// SIMATIC S7-200 SMART project (STEP 7-Micro/WIN SMART), CPU ST40

SYMBOL_TABLE 用户定义1
传感器1             I0.0
传感器2             I0.1
传感器3             I0.2
传感器4             I0.3
传感器5             I0.4
传感器6             I0.5
传感器7             I0.6
传感器8             I0.7
END_SYMBOL_TABLE

SYMBOL_TABLE 系统符号
Always_On        SM0.0    // 始终接通
First_Scan_On    SM0.1    // 仅在第一个扫描周期时接通
P0_Config        SMB30    // 组态端口 0 通信：奇偶校验、每个字符的数据位数、波特率和协议
END_SYMBOL_TABLE

SYMBOL_TABLE 表格 3
State            VB5000
SendBuffer       VB5100
RecvBuffer       VB5300
RecvLenth        VW5004
SendLenth        VW5006
SendBufferW      VW5100
RecvBufferW      VW5300
StateConnect     1
StateConnectWait 2
StateTransmit    3
StateTransmitWait 4
StateReceive     5
StateRecvCheck   6
StateDisconnect  7
StateDisconnectWait 8
ExitSwitch       10
SendLenthB       VB5008
END_SYMBOL_TABLE

ORGANIZATION_BLOCK 主程序:OB1
TITLE=程序注释
BEGIN
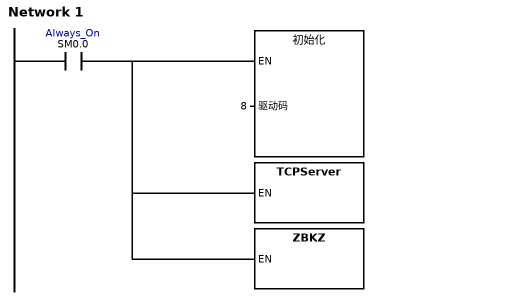
Network 1
LD     Always_On:SM0.0
CALL   初始化:SBR0, 8
CALL   TCPServer:SBR80
CALL   ZBKZ:SBR29
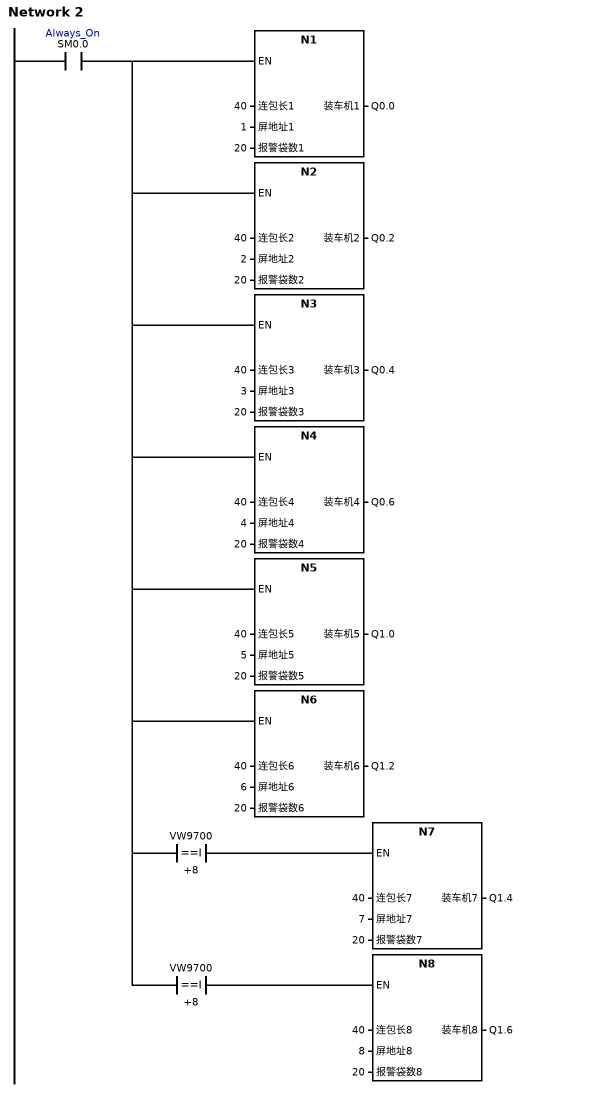
Network 2
LD     Always_On:SM0.0
LPS
CALL   N1:SBR1, 40, 1, 20, Q0.0
CALL   N2:SBR2, 40, 2, 20, Q0.2
CALL   N3:SBR3, 40, 3, 20, Q0.4
CALL   N4:SBR4, 40, 4, 20, Q0.6
CALL   N5:SBR5, 40, 5, 20, Q1.0
CALL   N6:SBR6, 40, 6, 20, Q1.2
AW=    VW9700, +8
CALL   N7:SBR7, 40, 7, 20, Q1.4
LPP
AW=    VW9700, +8
CALL   N8:SBR8, 40, 8, 20, Q1.6
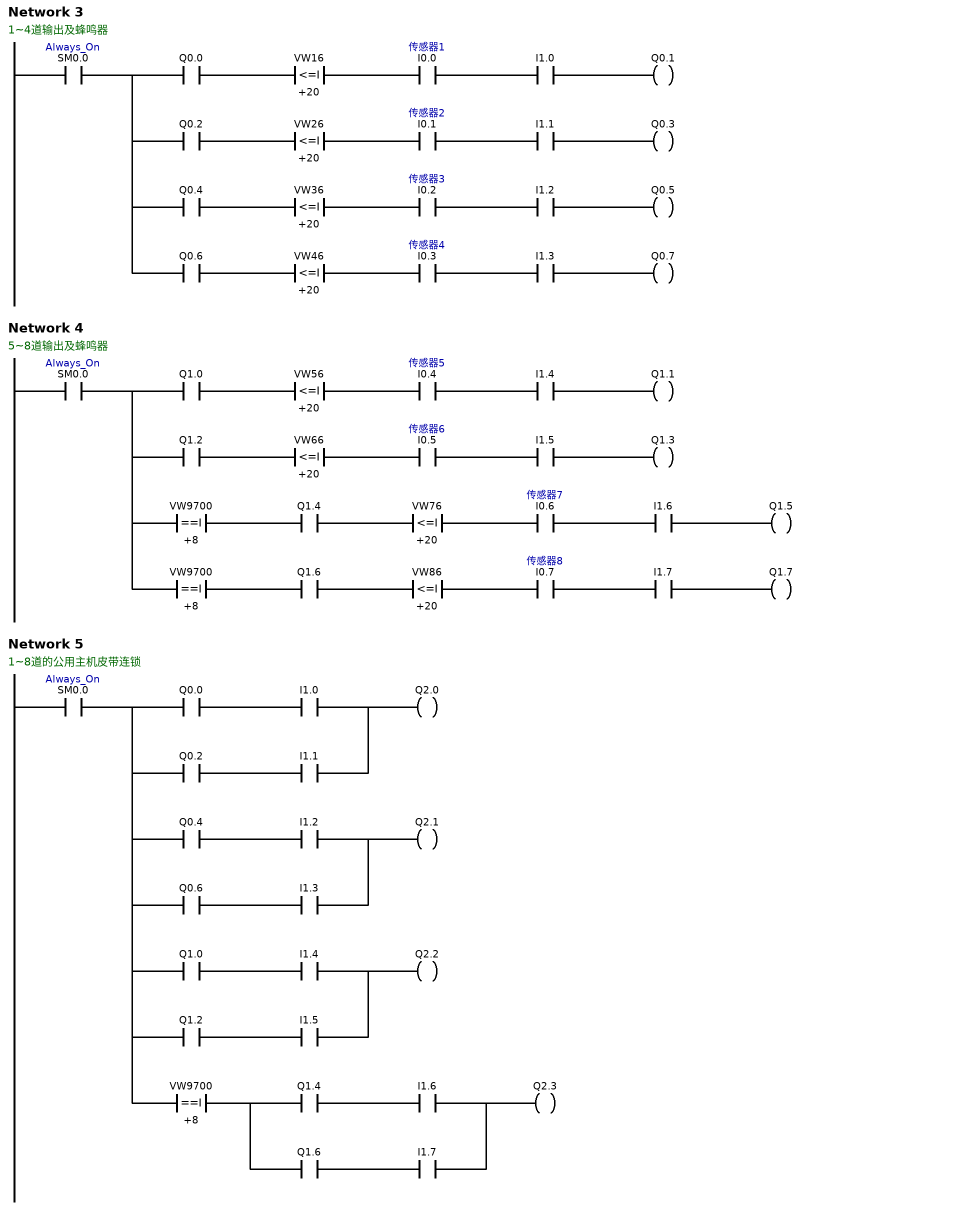
Network 3
// 1~4道输出及蜂鸣器
LD     Always_On:SM0.0
LPS
A      Q0.0
AW<=   VW16, +20
A      传感器1:I0.0
A      I1.0
=      Q0.1
LRD
A      Q0.2
AW<=   VW26, +20
A      传感器2:I0.1
A      I1.1
=      Q0.3
LRD
A      Q0.4
AW<=   VW36, +20
A      传感器3:I0.2
A      I1.2
=      Q0.5
LPP
A      Q0.6
AW<=   VW46, +20
A      传感器4:I0.3
A      I1.3
=      Q0.7
Network 4
// 5~8道输出及蜂鸣器
LD     Always_On:SM0.0
LPS
A      Q1.0
AW<=   VW56, +20
A      传感器5:I0.4
A      I1.4
=      Q1.1
LRD
A      Q1.2
AW<=   VW66, +20
A      传感器6:I0.5
A      I1.5
=      Q1.3
LRD
AW=    VW9700, +8
A      Q1.4
AW<=   VW76, +20
A      传感器7:I0.6
A      I1.6
=      Q1.5
LPP
AW=    VW9700, +8
A      Q1.6
AW<=   VW86, +20
A      传感器8:I0.7
A      I1.7
=      Q1.7
Network 5
// 1~8道的公用主机皮带连锁
LD     Always_On:SM0.0
LPS
LD     Q0.0
A      I1.0
LD     Q0.2
A      I1.1
OLD
ALD
=      Q2.0
LRD
LD     Q0.4
A      I1.2
LD     Q0.6
A      I1.3
OLD
ALD
=      Q2.1
LRD
LD     Q1.0
A      I1.4
LD     Q1.2
A      I1.5
OLD
ALD
=      Q2.2
LPP
AW=    VW9700, +8
LD     Q1.4
A      I1.6
LD     Q1.6
A      I1.7
OLD
ALD
=      Q2.3
END_ORGANIZATION_BLOCK

SUBROUTINE_BLOCK 初始化:SBR0
TITLE=子程序注释
VAR_INPUT
驱动码:WORD;	// LW0 
END_VAR
VAR
temp1:WORD;	// LW2 
temp2:WORD;	// LW4 
END_VAR
BEGIN
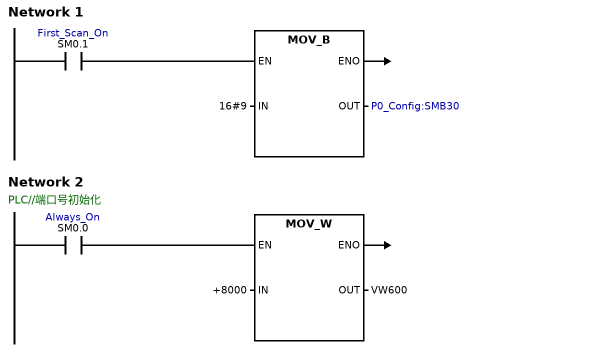
Network 1
// 首次扫描时，
// 初始化自由端口：
// - 选择9600波特
// - 选择8个数据位
// - 选择无校验
// 初始化RCV信息控制字节：
// - RCV被启用
// - 检测到信息字符结束
// - 将空闲行条件检测为
// 信息开始条件。
// 将信息字符结束设为hex OA（换行符）。
// 将空闲行超时设为5毫秒。
// 将最大字符数设为100。
// 为端口0在VB100位置启用带缓冲区的接收方框
LD     First_Scan_On:SM0.1
MOVB   16#9, P0_Config:SMB30
Network 2
// PLC//端口号初始化
LD     Always_On:SM0.0
MOVW   +8000, VW600
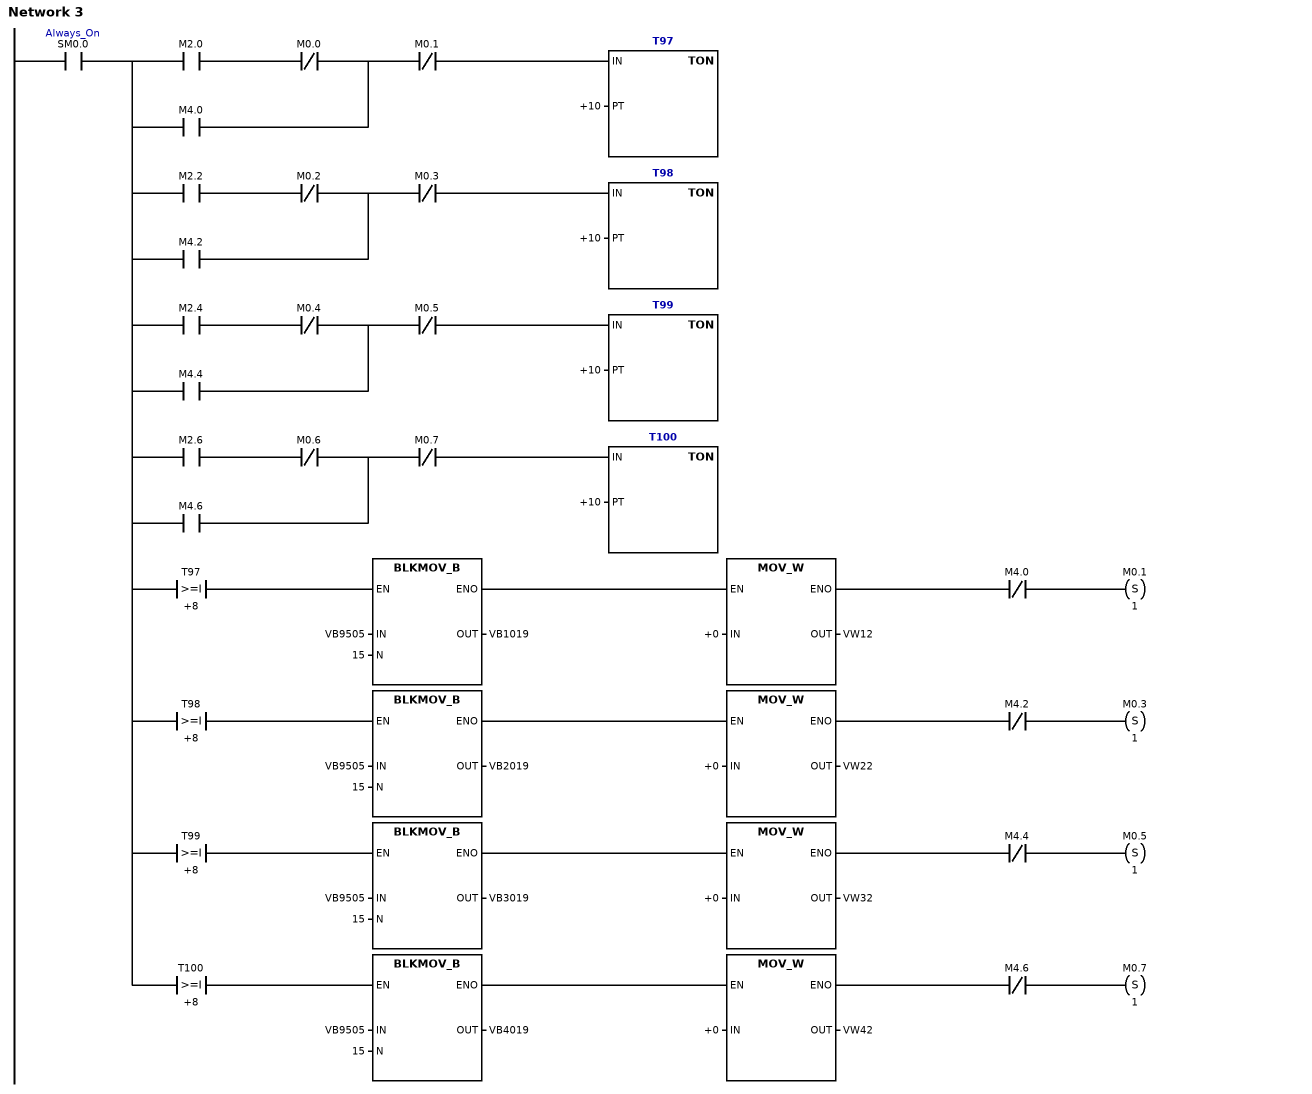
Network 3
LD     Always_On:SM0.0
LPS
LD     M2.0
AN     M0.0
O      M4.0
ALD
AN     M0.1
TON    T97, +10
LRD
LD     M2.2
AN     M0.2
O      M4.2
ALD
AN     M0.3
TON    T98, +10
LRD
LD     M2.4
AN     M0.4
O      M4.4
ALD
AN     M0.5
TON    T99, +10
LRD
LD     M2.6
AN     M0.6
O      M4.6
ALD
AN     M0.7
TON    T100, +10
LPP
LPS
AW>=   T97, +8
BMB    VB9505, VB1019, 15
AENO
MOVW   +0, VW12
AENO
AN     M4.0
S      M0.1, 1
LRD
AW>=   T98, +8
BMB    VB9505, VB2019, 15
AENO
MOVW   +0, VW22
AENO
AN     M4.2
S      M0.3, 1
LRD
AW>=   T99, +8
BMB    VB9505, VB3019, 15
AENO
MOVW   +0, VW32
AENO
AN     M4.4
S      M0.5, 1
LPP
AW>=   T100, +8
BMB    VB9505, VB4019, 15
AENO
MOVW   +0, VW42
AENO
AN     M4.6
S      M0.7, 1
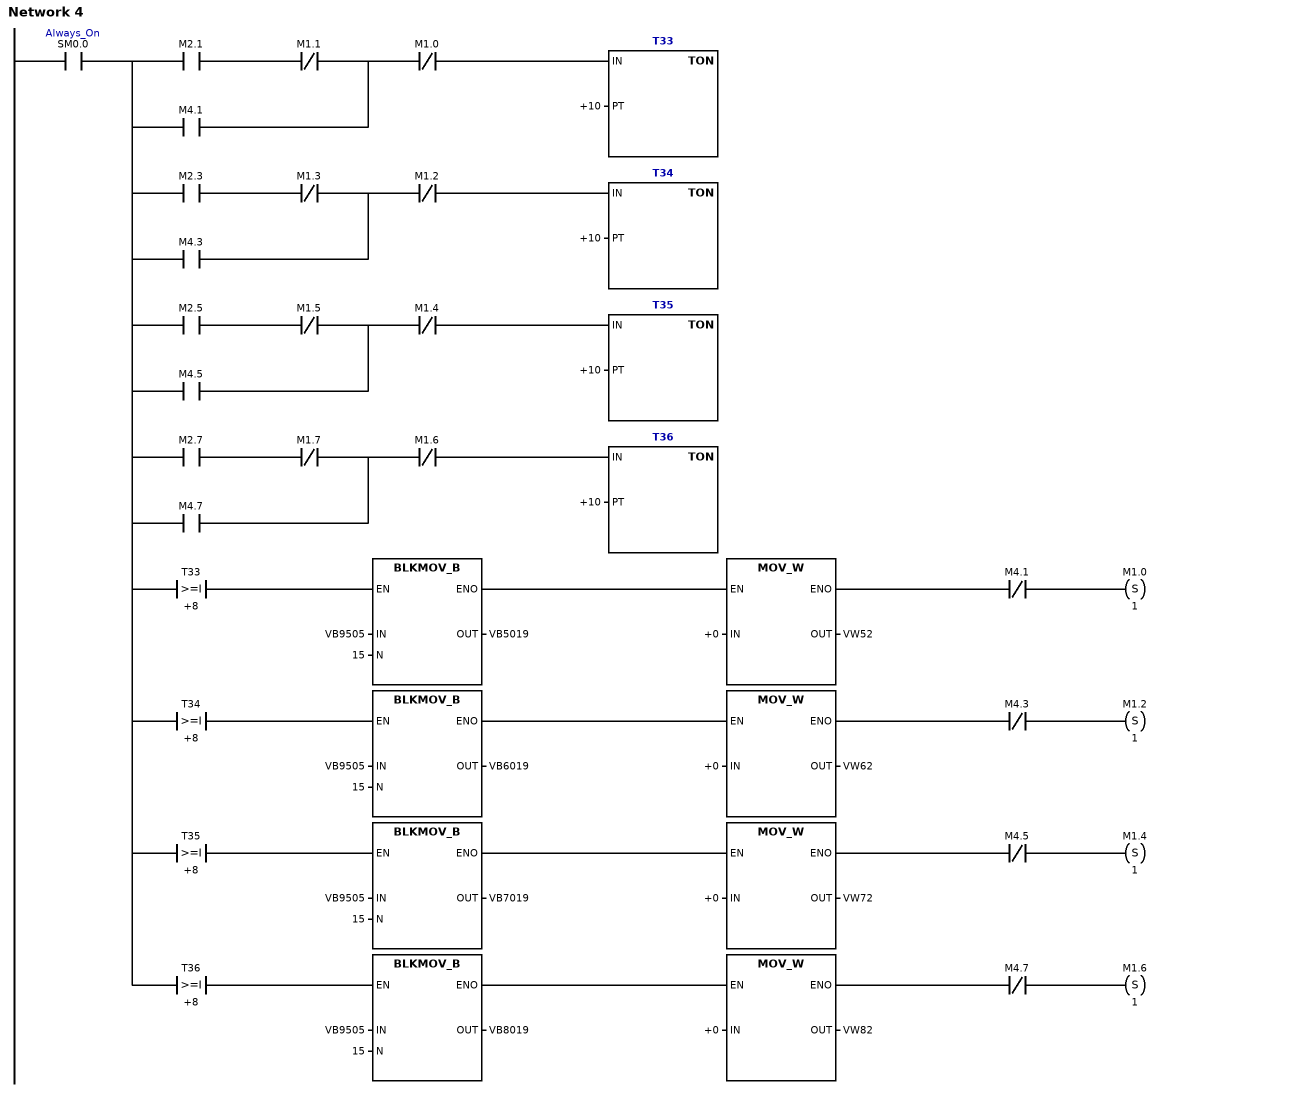
Network 4
LD     Always_On:SM0.0
LPS
LD     M2.1
AN     M1.1
O      M4.1
ALD
AN     M1.0
TON    T33, +10
LRD
LD     M2.3
AN     M1.3
O      M4.3
ALD
AN     M1.2
TON    T34, +10
LRD
LD     M2.5
AN     M1.5
O      M4.5
ALD
AN     M1.4
TON    T35, +10
LRD
LD     M2.7
AN     M1.7
O      M4.7
ALD
AN     M1.6
TON    T36, +10
LPP
LPS
AW>=   T33, +8
BMB    VB9505, VB5019, 15
AENO
MOVW   +0, VW52
AENO
AN     M4.1
S      M1.0, 1
LRD
AW>=   T34, +8
BMB    VB9505, VB6019, 15
AENO
MOVW   +0, VW62
AENO
AN     M4.3
S      M1.2, 1
LRD
AW>=   T35, +8
BMB    VB9505, VB7019, 15
AENO
MOVW   +0, VW72
AENO
AN     M4.5
S      M1.4, 1
LPP
AW>=   T36, +8
BMB    VB9505, VB8019, 15
AENO
MOVW   +0, VW82
AENO
AN     M4.7
S      M1.6, 1
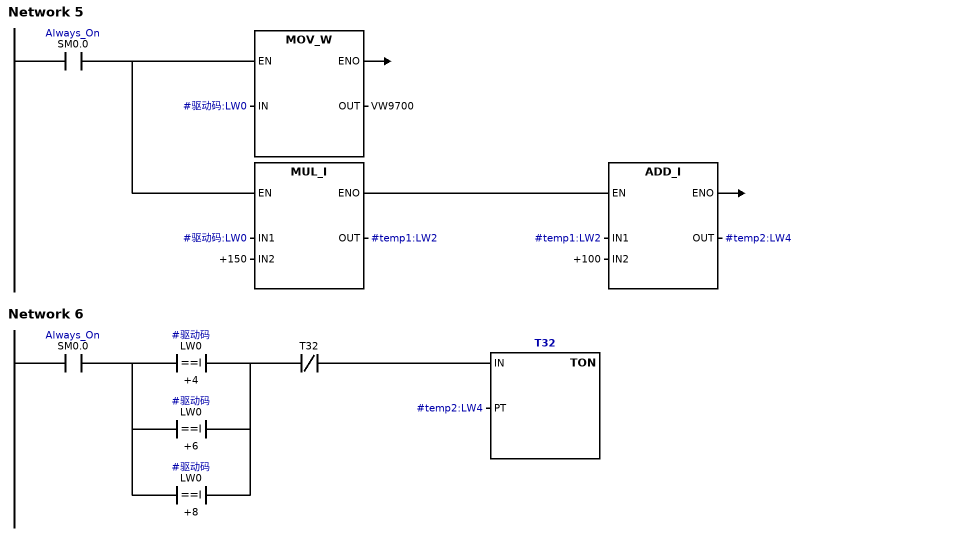
Network 5
LD     Always_On:SM0.0
MOVW   #驱动码:LW0, VW9700
MOVW   #驱动码:LW0, #temp1:LW2
AENO
*I     +150, #temp1:LW2
AENO
MOVW   #temp1:LW2, #temp2:LW4
+I     +100, #temp2:LW4
Network 6
LD     Always_On:SM0.0
LDW=   #驱动码:LW0, +4
OW=    #驱动码:LW0, +6
OW=    #驱动码:LW0, +8
ALD
AN     T32
TON    T32, #temp2:LW4
END_SUBROUTINE_BLOCK

SUBROUTINE_BLOCK N1:SBR1
TITLE=
VAR_INPUT
连包长1:WORD;	// LW0 
屏地址1:BYTE;	// LB2 
报警袋数1:WORD;	// LW3 
END_VAR
VAR_OUTPUT
装车机1:BOOL;	// L5.0 
END_VAR
VAR
总袋数1:WORD;	// LW6 
袋长1:WORD;	// LW8 
已装袋数1:WORD;	// LW10 
剩余袋数1:WORD;	// LW12 
END_VAR
BEGIN
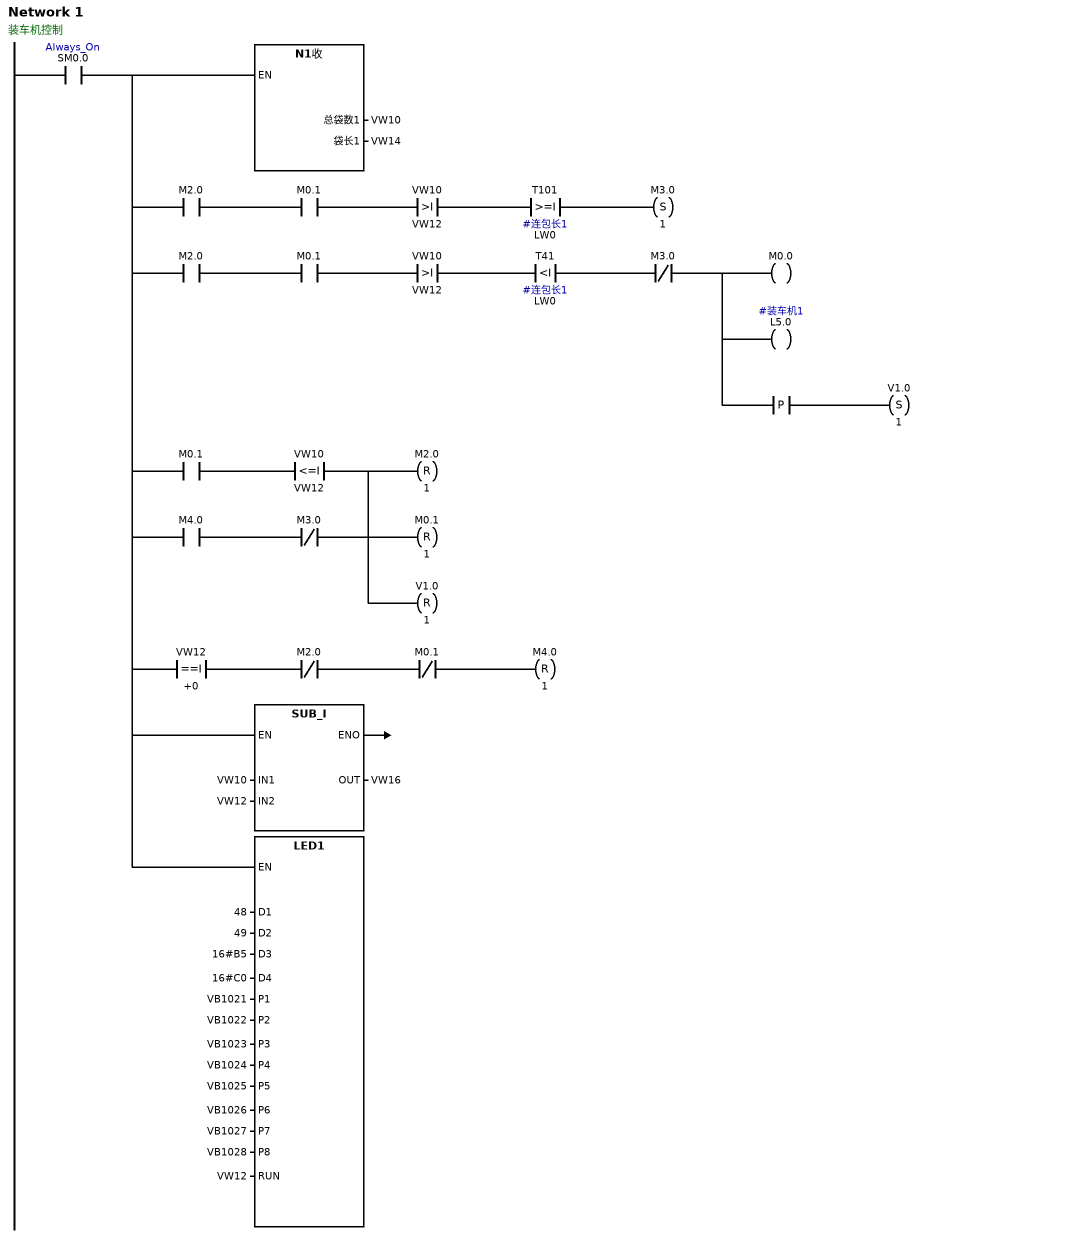
Network 1
// 装车机控制
LD     Always_On:SM0.0
LPS
CALL   N1收:SBR21, VW10, VW14
A      M2.0
A      M0.1
AW>    VW10, VW12
AW>=   T101, #连包长1:LW0
S      M3.0, 1
LRD
A      M2.0
A      M0.1
AW>    VW10, VW12
AW<    T41, #连包长1:LW0
AN     M3.0
=      M0.0
=      #装车机1:L5.0
EU
S      V1.0, 1
LRD
LD     M0.1
AW<=   VW10, VW12
LD     M4.0
AN     M3.0
OLD
ALD
R      M2.0, 1
R      M0.1, 1
R      V1.0, 1
LPP
LPS
AW=    VW12, +0
AN     M2.0
AN     M0.1
R      M4.0, 1
LRD
MOVW   VW10, VW16
-I     VW12, VW16
LPP
CALL   LED1:SBR11, 48, 49, 16#B5, 16#C0, VB1021, VB1022, VB1023, VB1024, VB1025, VB1026, VB1027, VB1028, VW12
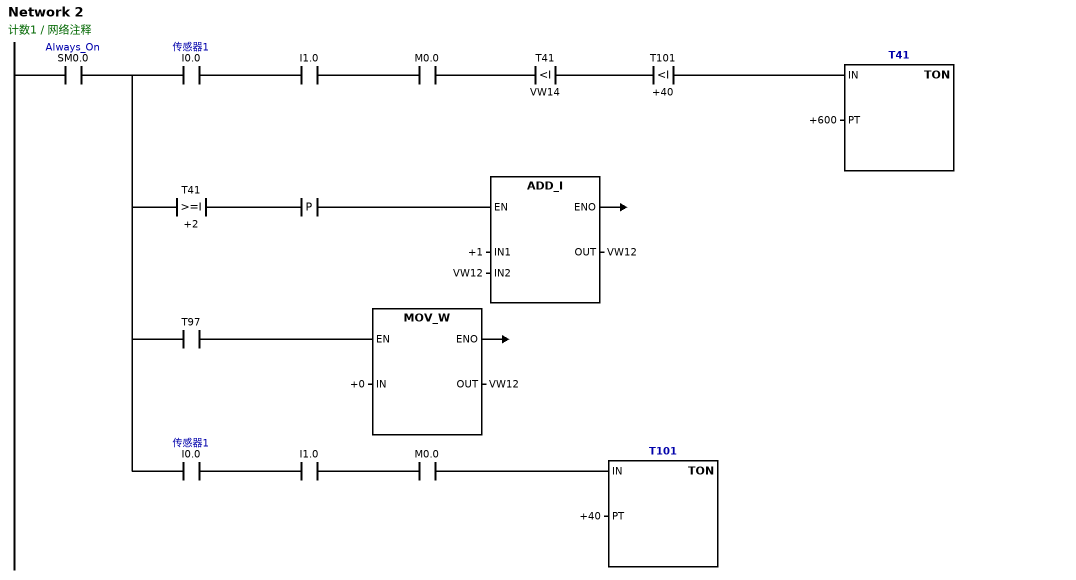
Network 2
// 计数1
// 网络注释
LD     Always_On:SM0.0
LPS
A      传感器1:I0.0
A      I1.0
A      M0.0
AW<    T41, VW14
AW<    T101, +40
TON    T41, +600
LRD
AW>=   T41, +2
EU
+I     +1, VW12
LRD
A      T97
MOVW   +0, VW12
LPP
A      传感器1:I0.0
A      I1.0
A      M0.0
TON    T101, +40
END_SUBROUTINE_BLOCK

SUBROUTINE_BLOCK N2:SBR2
TITLE=
VAR_INPUT
连包长2:WORD;	// LW0 
屏地址2:BYTE;	// LB2 
报警袋数2:WORD;	// LW3 
END_VAR
VAR_OUTPUT
装车机2:BOOL;	// L5.0 
END_VAR
VAR
总袋数2:WORD;	// LW6 
袋长2:WORD;	// LW8 
已装袋数2:WORD;	// LW10 
剩余袋数2:WORD;	// LW12 
END_VAR
BEGIN
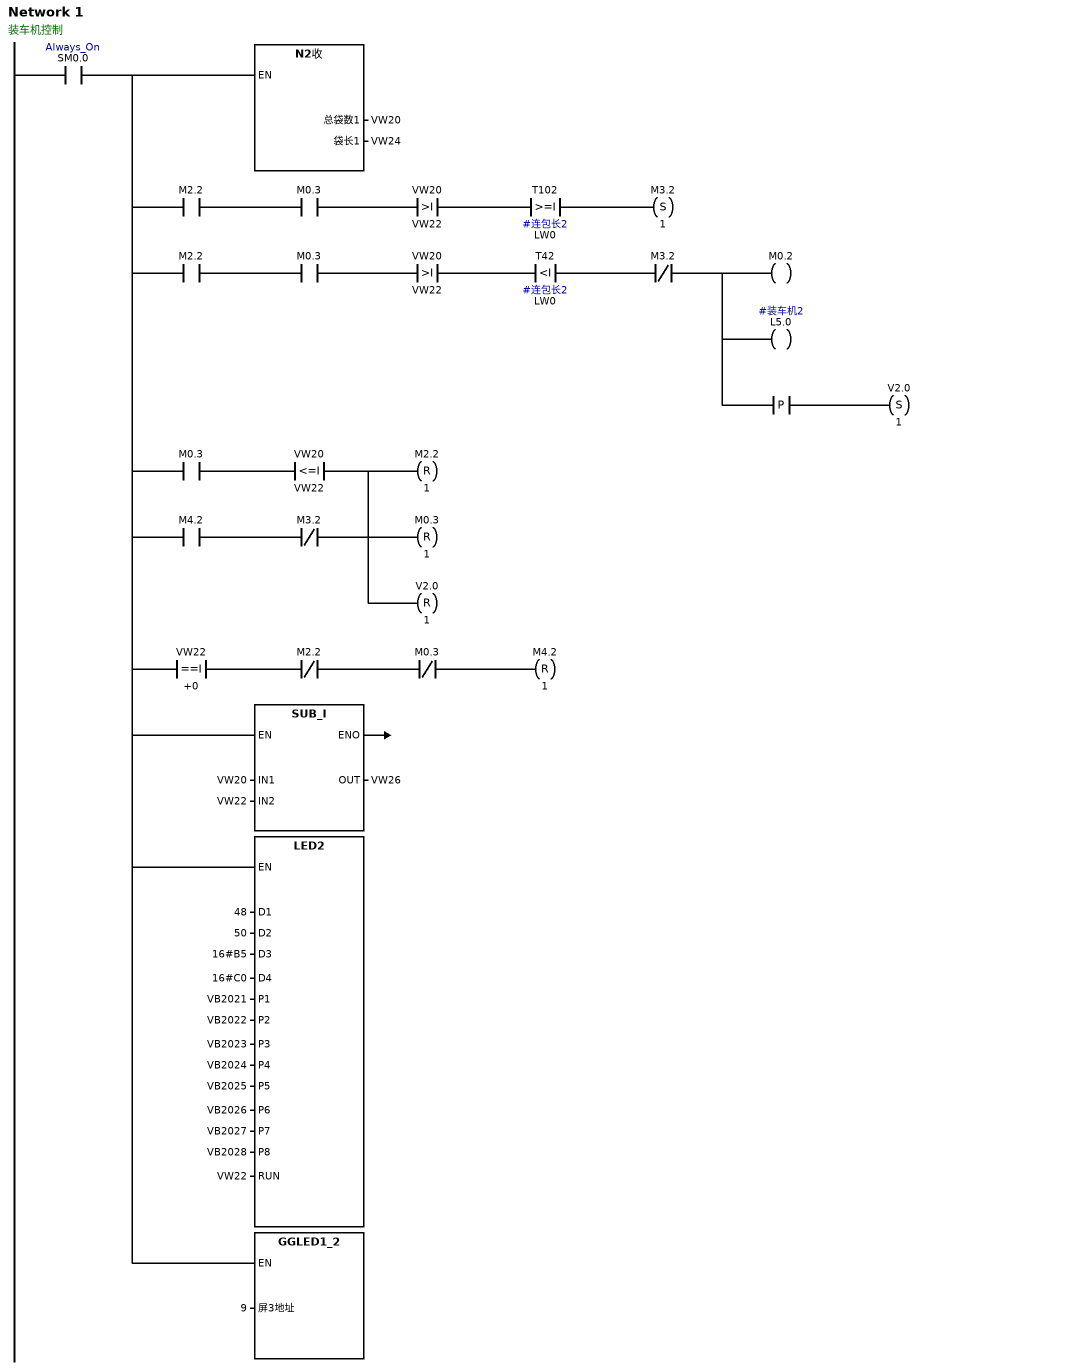
Network 1
// 装车机控制
LD     Always_On:SM0.0
LPS
CALL   N2收:SBR22, VW20, VW24
A      M2.2
A      M0.3
AW>    VW20, VW22
AW>=   T102, #连包长2:LW0
S      M3.2, 1
LRD
A      M2.2
A      M0.3
AW>    VW20, VW22
AW<    T42, #连包长2:LW0
AN     M3.2
=      M0.2
=      #装车机2:L5.0
EU
S      V2.0, 1
LRD
LD     M0.3
AW<=   VW20, VW22
LD     M4.2
AN     M3.2
OLD
ALD
R      M2.2, 1
R      M0.3, 1
R      V2.0, 1
LPP
LPS
AW=    VW22, +0
AN     M2.2
AN     M0.3
R      M4.2, 1
LRD
MOVW   VW20, VW26
-I     VW22, VW26
LRD
CALL   LED2:SBR12, 48, 50, 16#B5, 16#C0, VB2021, VB2022, VB2023, VB2024, VB2025, VB2026, VB2027, VB2028, VW22
LPP
CALL   GGLED1_2:SBR31, 9
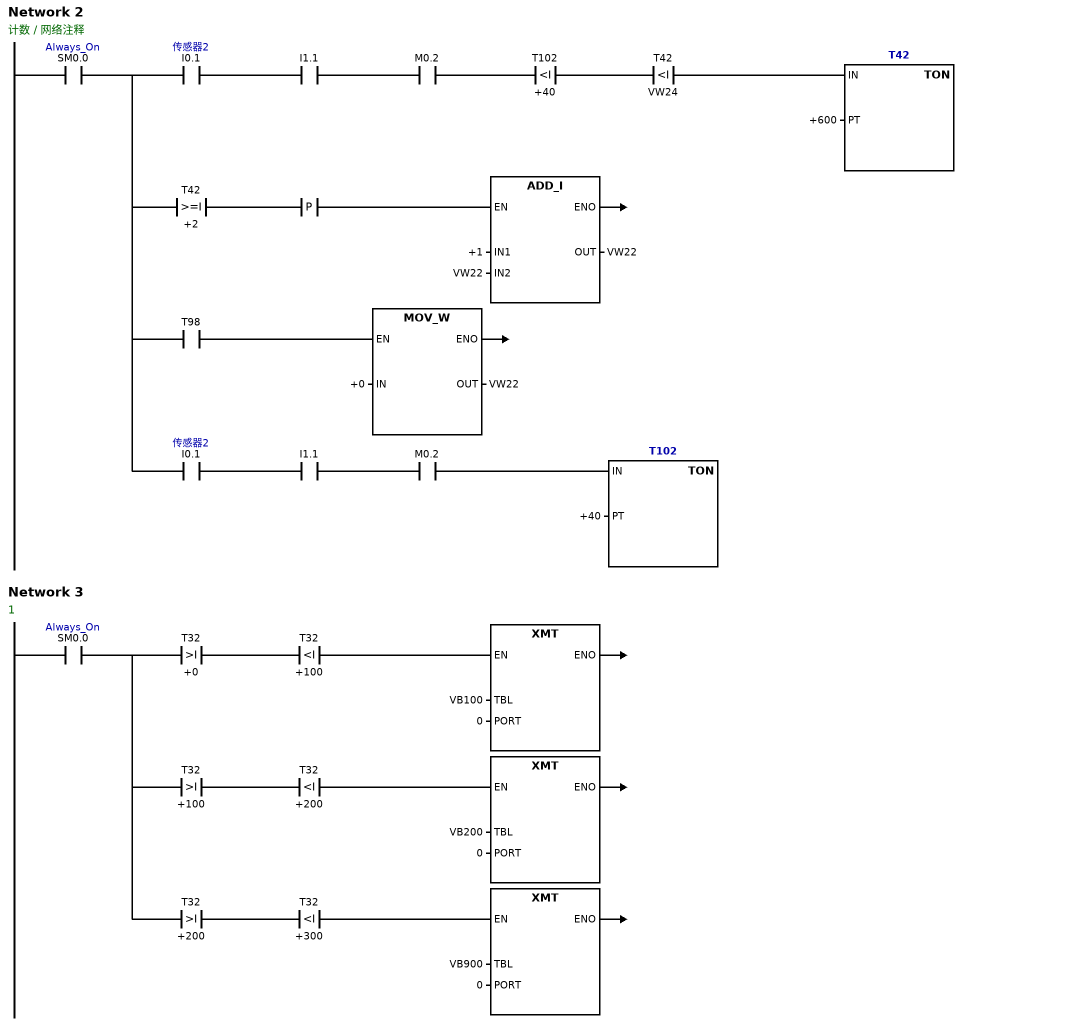
Network 2
// 计数
// 网络注释
LD     Always_On:SM0.0
LPS
A      传感器2:I0.1
A      I1.1
A      M0.2
AW<    T102, +40
AW<    T42, VW24
TON    T42, +600
LRD
AW>=   T42, +2
EU
+I     +1, VW22
LRD
A      T98
MOVW   +0, VW22
LPP
A      传感器2:I0.1
A      I1.1
A      M0.2
TON    T102, +40
Network 3
// 1
LD     Always_On:SM0.0
LPS
AW>    T32, +0
AW<    T32, +100
XMT    VB100, 0
LRD
AW>    T32, +100
AW<    T32, +200
XMT    VB200, 0
LPP
AW>    T32, +200
AW<    T32, +300
XMT    VB900, 0
END_SUBROUTINE_BLOCK

SUBROUTINE_BLOCK N3:SBR3
TITLE=
VAR_INPUT
连包长3:WORD;	// LW0 
屏地址3:BYTE;	// LB2 
报警袋数3:WORD;	// LW3 
END_VAR
VAR_OUTPUT
装车机3:BOOL;	// L5.0 
END_VAR
VAR
总袋数3:WORD;	// LW6 
袋长3:WORD;	// LW8 
已装袋数3:WORD;	// LW10 
剩余袋数3:WORD;	// LW12 
END_VAR
BEGIN
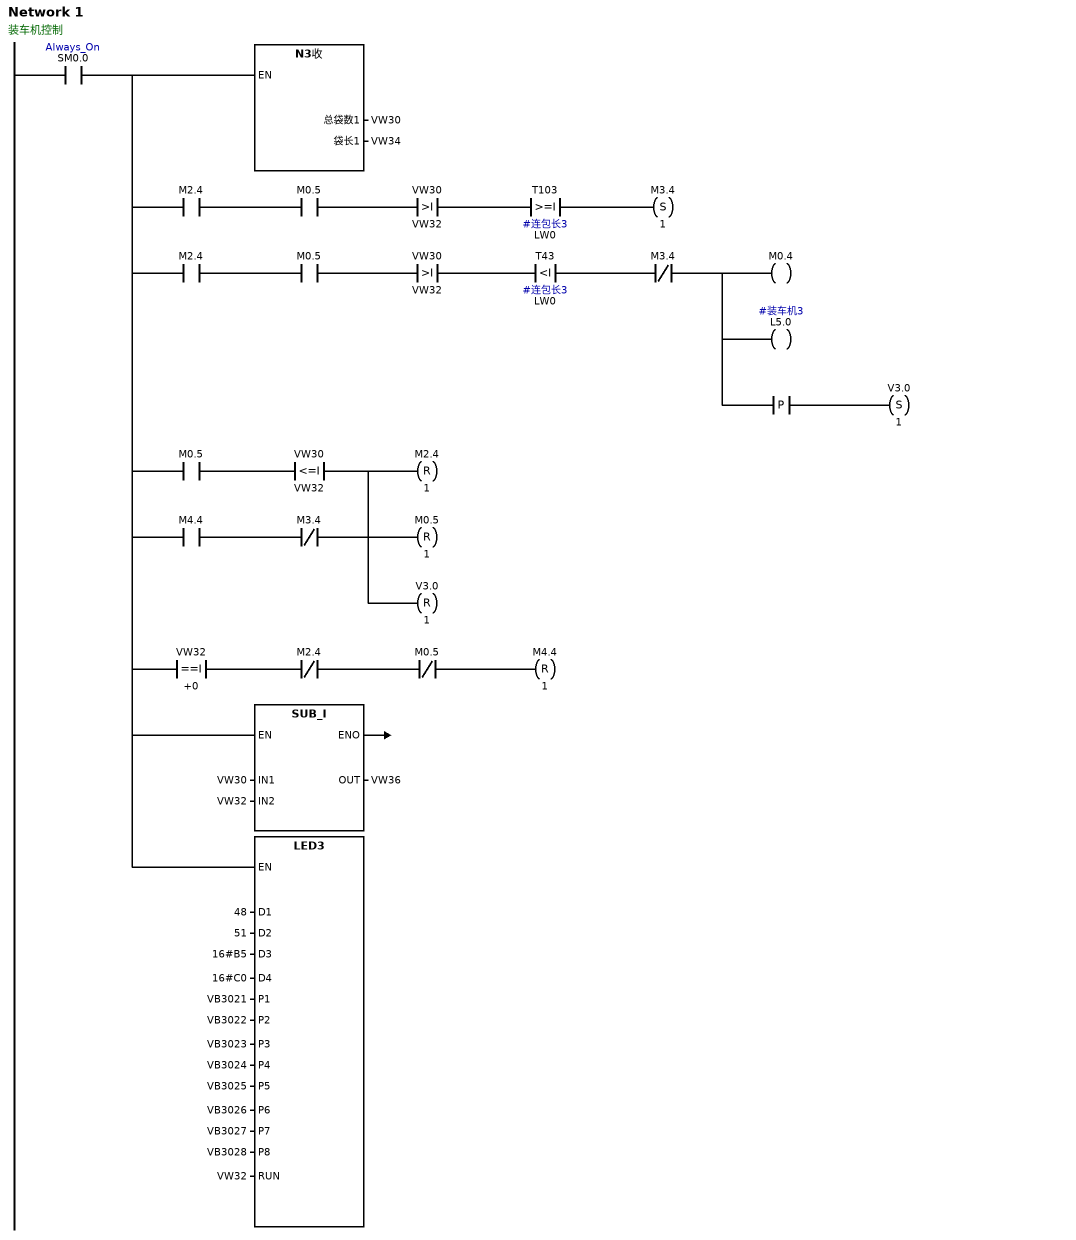
Network 1
// 装车机控制
LD     Always_On:SM0.0
LPS
CALL   N3收:SBR23, VW30, VW34
A      M2.4
A      M0.5
AW>    VW30, VW32
AW>=   T103, #连包长3:LW0
S      M3.4, 1
LRD
A      M2.4
A      M0.5
AW>    VW30, VW32
AW<    T43, #连包长3:LW0
AN     M3.4
=      M0.4
=      #装车机3:L5.0
EU
S      V3.0, 1
LRD
LD     M0.5
AW<=   VW30, VW32
LD     M4.4
AN     M3.4
OLD
ALD
R      M2.4, 1
R      M0.5, 1
R      V3.0, 1
LPP
LPS
AW=    VW32, +0
AN     M2.4
AN     M0.5
R      M4.4, 1
LRD
MOVW   VW30, VW36
-I     VW32, VW36
LPP
CALL   LED3:SBR13, 48, 51, 16#B5, 16#C0, VB3021, VB3022, VB3023, VB3024, VB3025, VB3026, VB3027, VB3028, VW32
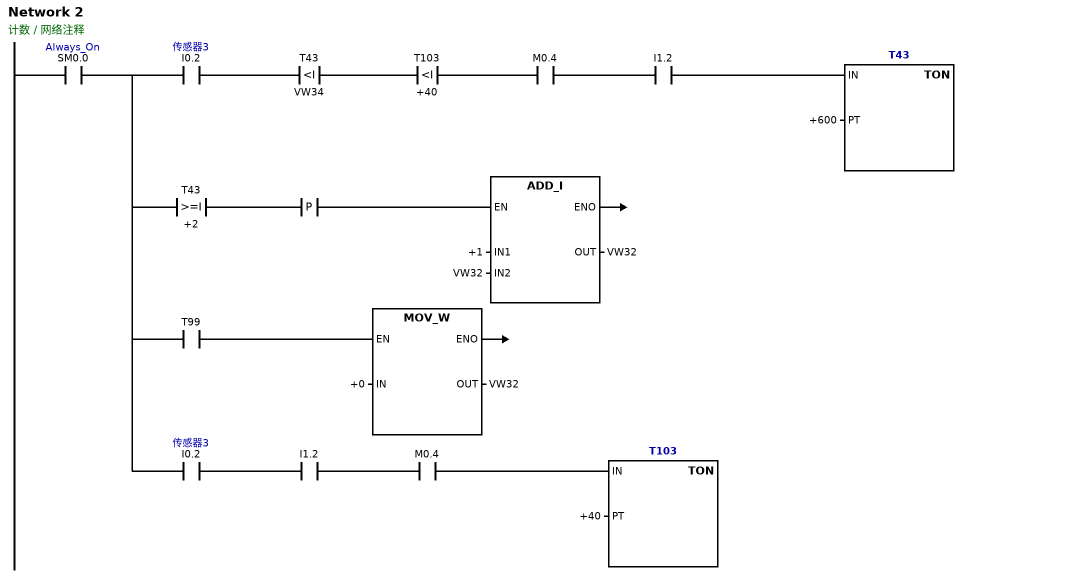
Network 2
// 计数
// 网络注释
LD     Always_On:SM0.0
LPS
A      传感器3:I0.2
AW<    T43, VW34
AW<    T103, +40
A      M0.4
A      I1.2
TON    T43, +600
LRD
AW>=   T43, +2
EU
+I     +1, VW32
LRD
A      T99
MOVW   +0, VW32
LPP
A      传感器3:I0.2
A      I1.2
A      M0.4
TON    T103, +40
END_SUBROUTINE_BLOCK

SUBROUTINE_BLOCK N4:SBR4
TITLE=
VAR_INPUT
连包长4:WORD;	// LW0 
屏地址4:BYTE;	// LB2 
报警袋数4:WORD;	// LW3 
END_VAR
VAR_OUTPUT
装车机4:BOOL;	// L5.0 
END_VAR
VAR
总袋数4:WORD;	// LW6 
袋长4:WORD;	// LW8 
已装袋数4:WORD;	// LW10 
剩余袋数4:WORD;	// LW12 
END_VAR
BEGIN
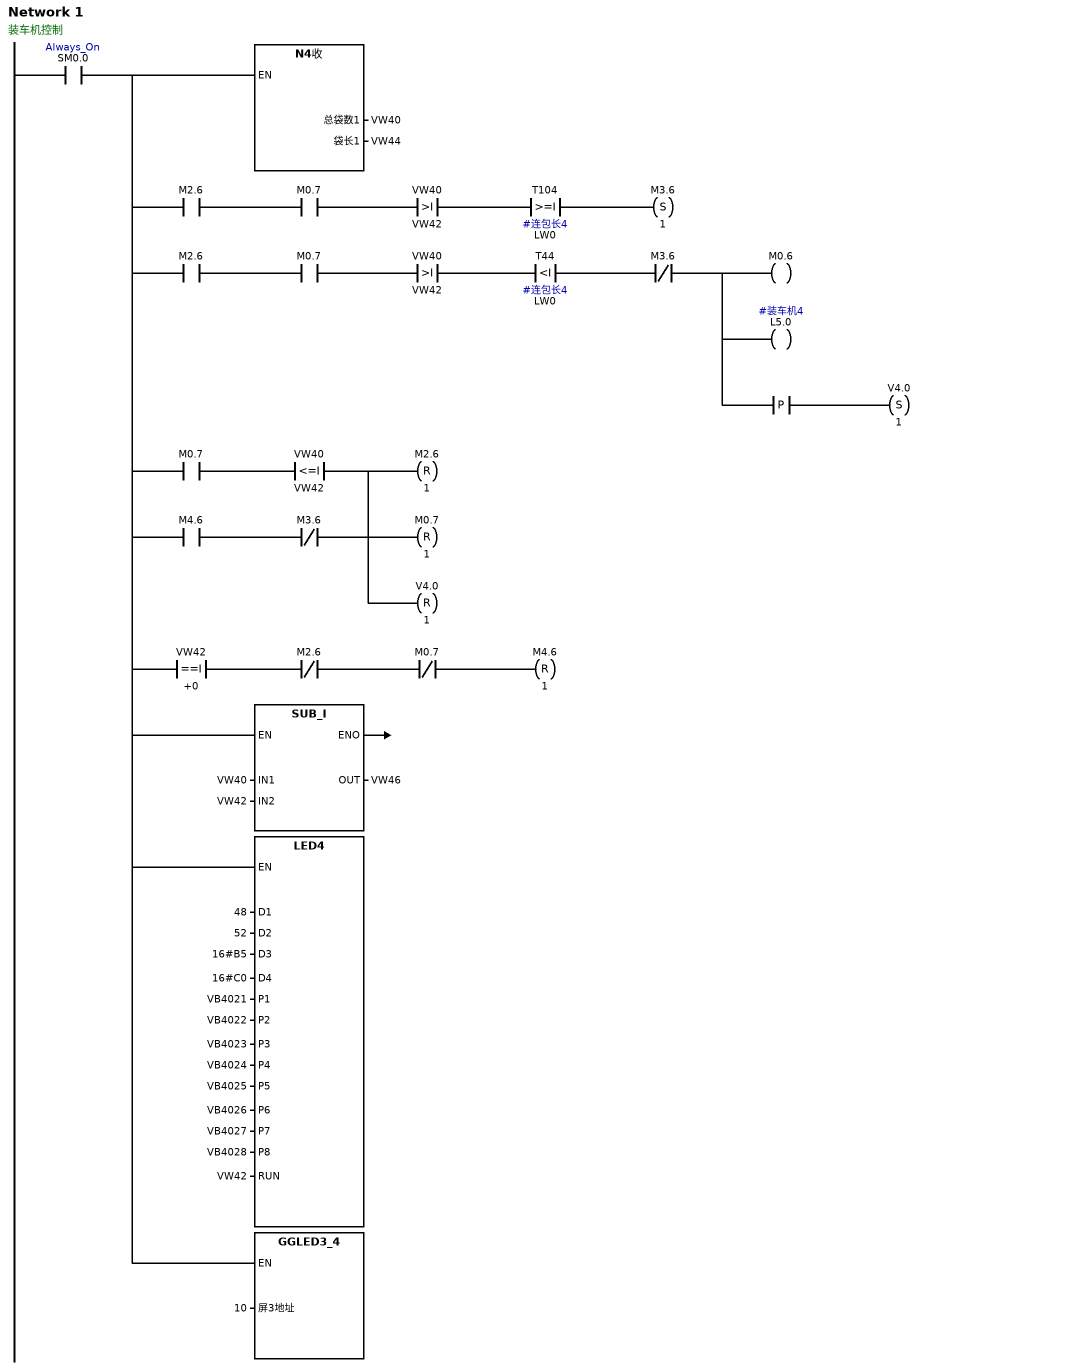
Network 1
// 装车机控制
LD     Always_On:SM0.0
LPS
CALL   N4收:SBR24, VW40, VW44
A      M2.6
A      M0.7
AW>    VW40, VW42
AW>=   T104, #连包长4:LW0
S      M3.6, 1
LRD
A      M2.6
A      M0.7
AW>    VW40, VW42
AW<    T44, #连包长4:LW0
AN     M3.6
=      M0.6
=      #装车机4:L5.0
EU
S      V4.0, 1
LRD
LD     M0.7
AW<=   VW40, VW42
LD     M4.6
AN     M3.6
OLD
ALD
R      M2.6, 1
R      M0.7, 1
R      V4.0, 1
LPP
LPS
AW=    VW42, +0
AN     M2.6
AN     M0.7
R      M4.6, 1
LRD
MOVW   VW40, VW46
-I     VW42, VW46
LRD
CALL   LED4:SBR14, 48, 52, 16#B5, 16#C0, VB4021, VB4022, VB4023, VB4024, VB4025, VB4026, VB4027, VB4028, VW42
LPP
CALL   GGLED3_4:SBR32, 10
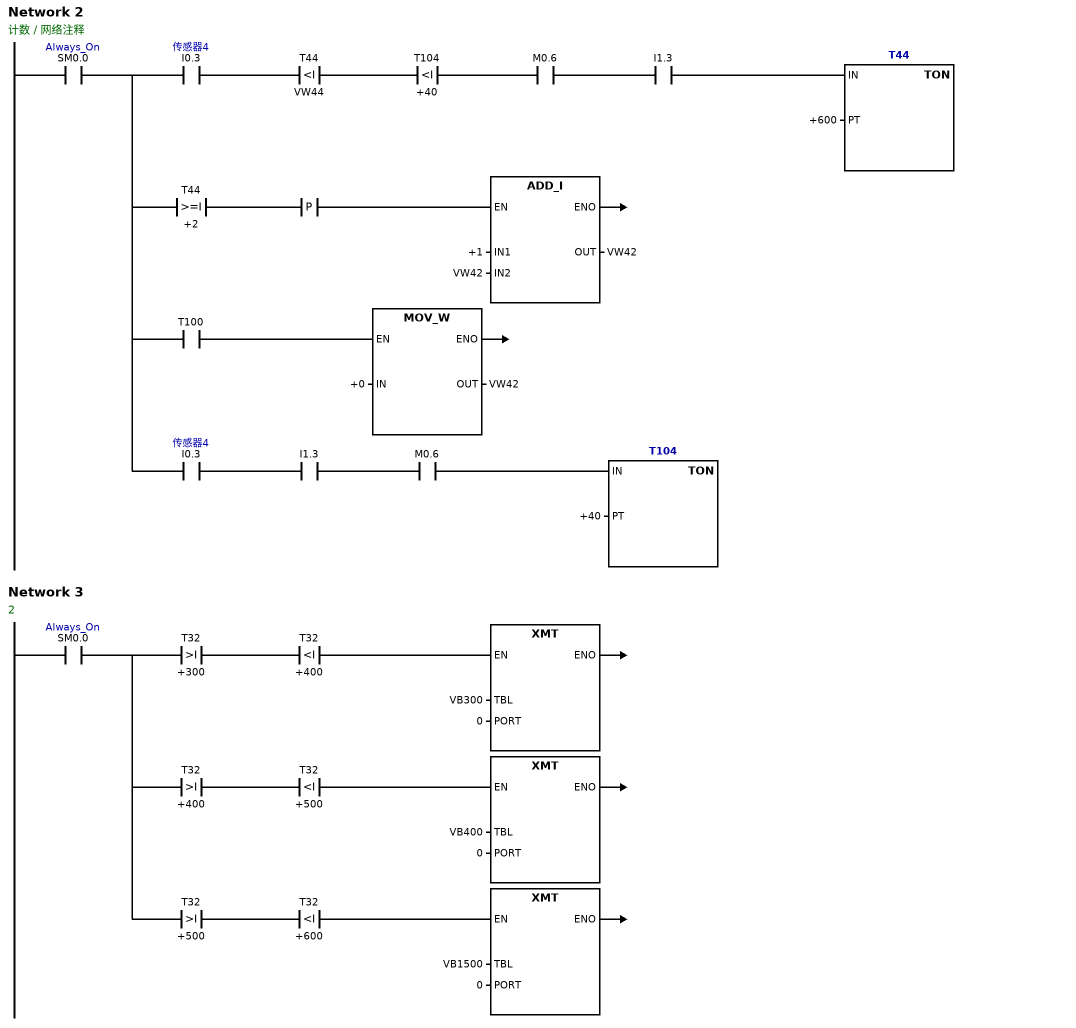
Network 2
// 计数
// 网络注释
LD     Always_On:SM0.0
LPS
A      传感器4:I0.3
AW<    T44, VW44
AW<    T104, +40
A      M0.6
A      I1.3
TON    T44, +600
LRD
AW>=   T44, +2
EU
+I     +1, VW42
LRD
A      T100
MOVW   +0, VW42
LPP
A      传感器4:I0.3
A      I1.3
A      M0.6
TON    T104, +40
Network 3
// 2
LD     Always_On:SM0.0
LPS
AW>    T32, +300
AW<    T32, +400
XMT    VB300, 0
LRD
AW>    T32, +400
AW<    T32, +500
XMT    VB400, 0
LPP
AW>    T32, +500
AW<    T32, +600
XMT    VB1500, 0
END_SUBROUTINE_BLOCK

SUBROUTINE_BLOCK N5:SBR5
TITLE=
VAR_INPUT
连包长5:WORD;	// LW0 
屏地址5:BYTE;	// LB2 
报警袋数5:WORD;	// LW3 
END_VAR
VAR_OUTPUT
装车机5:BOOL;	// L5.0 
END_VAR
VAR
总袋数5:WORD;	// LW6 
袋长5:WORD;	// LW8 
已装袋数5:WORD;	// LW10 
剩余袋数5:WORD;	// LW12 
END_VAR
BEGIN
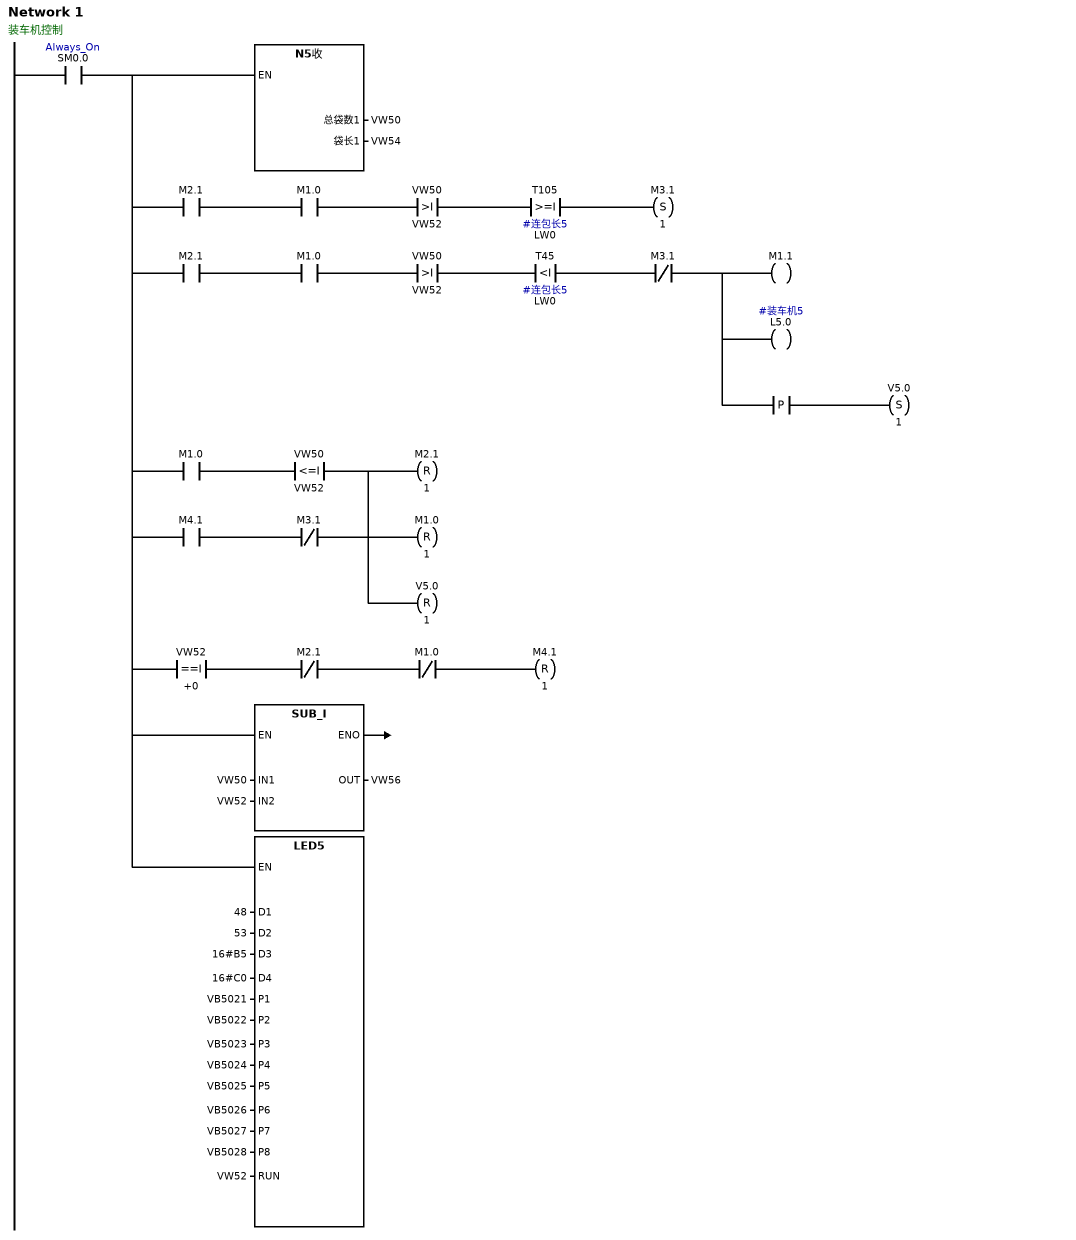
Network 1
// 装车机控制
LD     Always_On:SM0.0
LPS
CALL   N5收:SBR25, VW50, VW54
A      M2.1
A      M1.0
AW>    VW50, VW52
AW>=   T105, #连包长5:LW0
S      M3.1, 1
LRD
A      M2.1
A      M1.0
AW>    VW50, VW52
AW<    T45, #连包长5:LW0
AN     M3.1
=      M1.1
=      #装车机5:L5.0
EU
S      V5.0, 1
LRD
LD     M1.0
AW<=   VW50, VW52
LD     M4.1
AN     M3.1
OLD
ALD
R      M2.1, 1
R      M1.0, 1
R      V5.0, 1
LPP
LPS
AW=    VW52, +0
AN     M2.1
AN     M1.0
R      M4.1, 1
LRD
MOVW   VW50, VW56
-I     VW52, VW56
LPP
CALL   LED5:SBR15, 48, 53, 16#B5, 16#C0, VB5021, VB5022, VB5023, VB5024, VB5025, VB5026, VB5027, VB5028, VW52
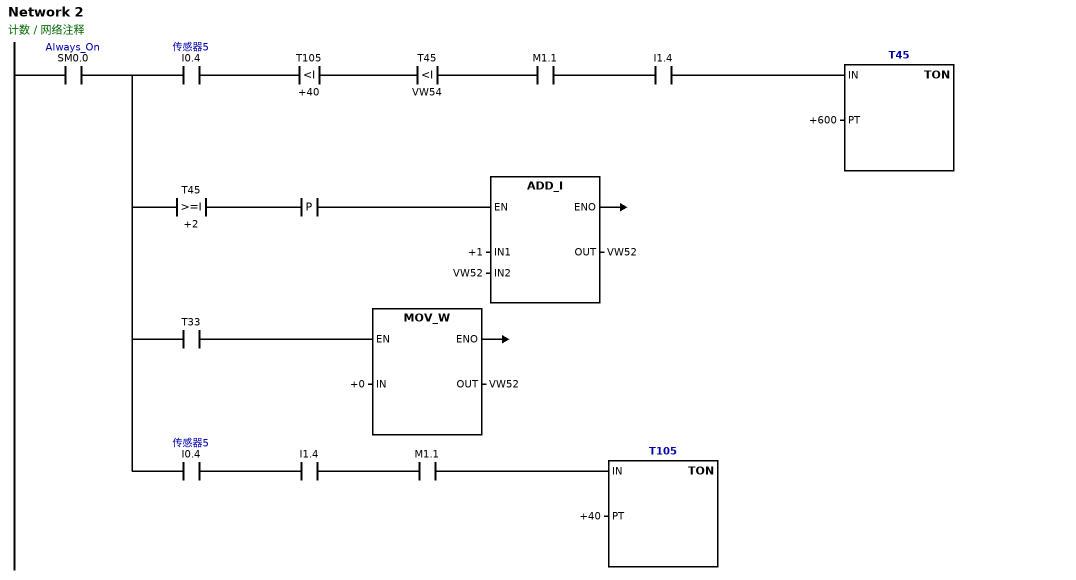
Network 2
// 计数
// 网络注释
LD     Always_On:SM0.0
LPS
A      传感器5:I0.4
AW<    T105, +40
AW<    T45, VW54
A      M1.1
A      I1.4
TON    T45, +600
LRD
AW>=   T45, +2
EU
+I     +1, VW52
LRD
A      T33
MOVW   +0, VW52
LPP
A      传感器5:I0.4
A      I1.4
A      M1.1
TON    T105, +40
END_SUBROUTINE_BLOCK

SUBROUTINE_BLOCK N6:SBR6
TITLE=
VAR_INPUT
连包长6:WORD;	// LW0 
屏地址6:BYTE;	// LB2 
报警袋数6:WORD;	// LW3 
END_VAR
VAR_OUTPUT
装车机6:BOOL;	// L5.0 
END_VAR
VAR
总袋数6:WORD;	// LW6 
袋长6:WORD;	// LW8 
已装袋数6:WORD;	// LW10 
剩余袋数6:WORD;	// LW12 
END_VAR
BEGIN
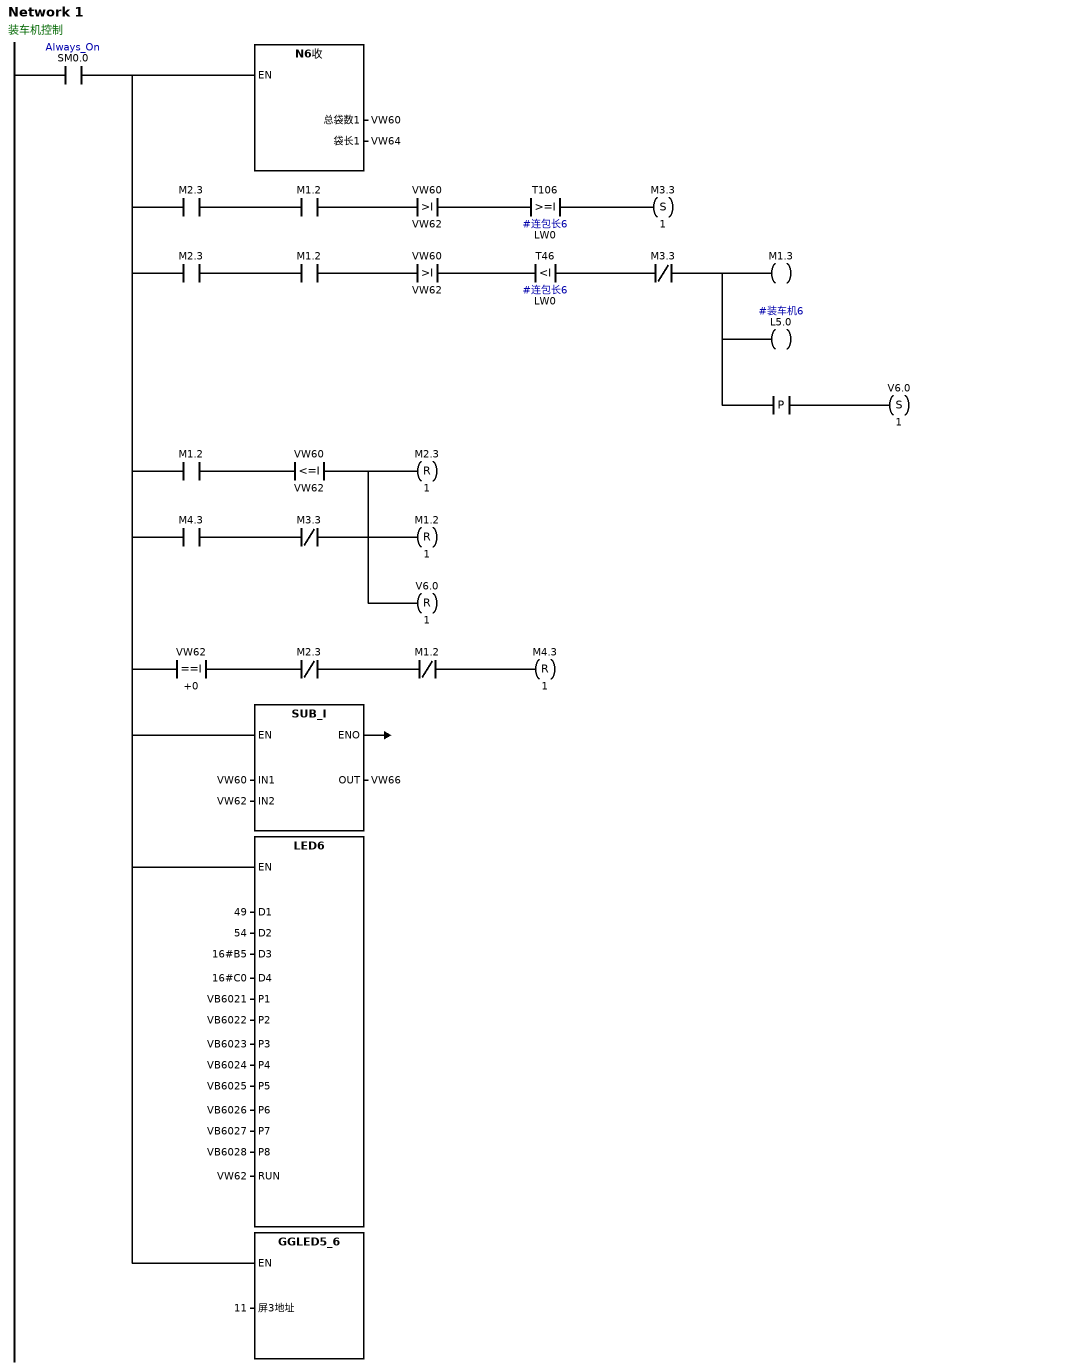
Network 1
// 装车机控制
LD     Always_On:SM0.0
LPS
CALL   N6收:SBR26, VW60, VW64
A      M2.3
A      M1.2
AW>    VW60, VW62
AW>=   T106, #连包长6:LW0
S      M3.3, 1
LRD
A      M2.3
A      M1.2
AW>    VW60, VW62
AW<    T46, #连包长6:LW0
AN     M3.3
=      M1.3
=      #装车机6:L5.0
EU
S      V6.0, 1
LRD
LD     M1.2
AW<=   VW60, VW62
LD     M4.3
AN     M3.3
OLD
ALD
R      M2.3, 1
R      M1.2, 1
R      V6.0, 1
LPP
LPS
AW=    VW62, +0
AN     M2.3
AN     M1.2
R      M4.3, 1
LRD
MOVW   VW60, VW66
-I     VW62, VW66
LRD
CALL   LED6:SBR16, 49, 54, 16#B5, 16#C0, VB6021, VB6022, VB6023, VB6024, VB6025, VB6026, VB6027, VB6028, VW62
LPP
CALL   GGLED5_6:SBR33, 11
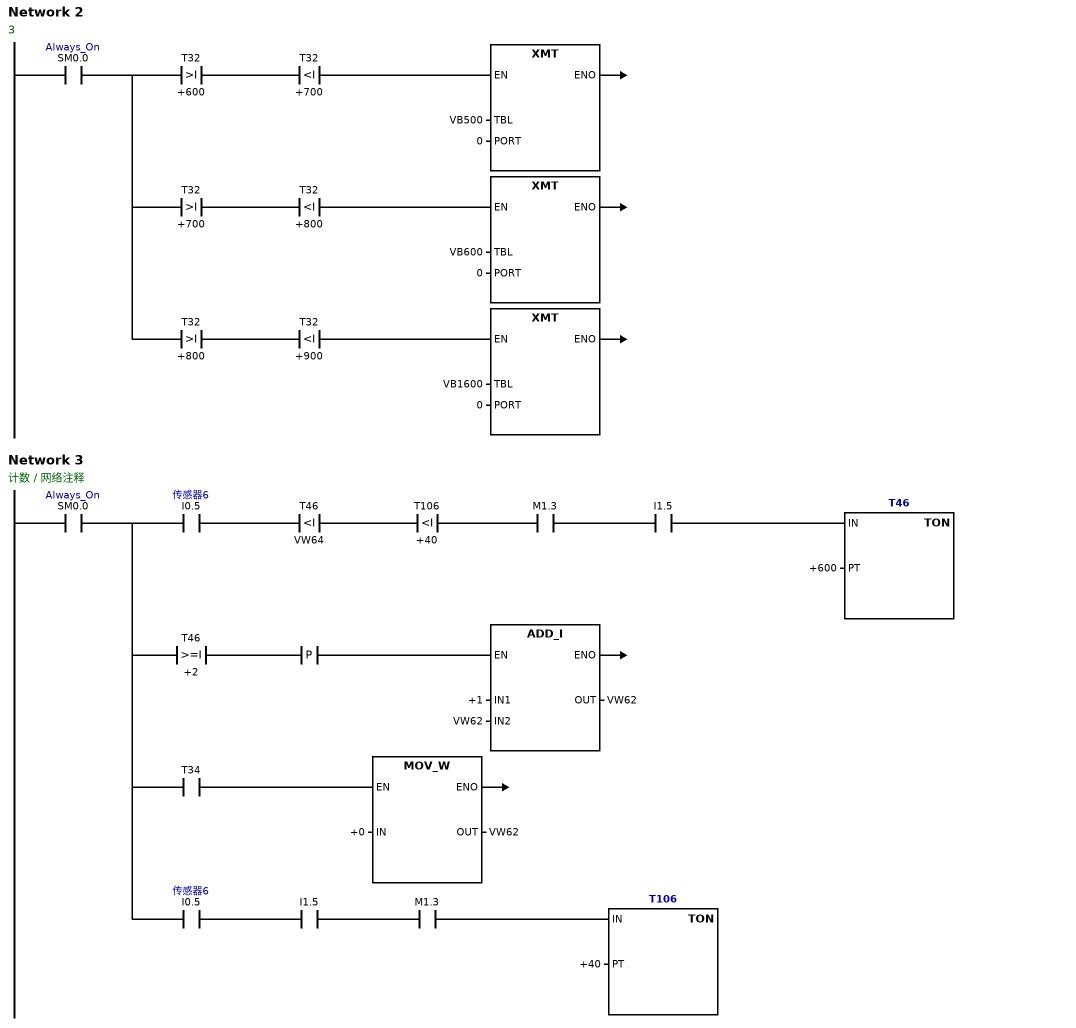
Network 2
// 3
LD     Always_On:SM0.0
LPS
AW>    T32, +600
AW<    T32, +700
XMT    VB500, 0
LRD
AW>    T32, +700
AW<    T32, +800
XMT    VB600, 0
LPP
AW>    T32, +800
AW<    T32, +900
XMT    VB1600, 0
Network 3
// 计数
// 网络注释
LD     Always_On:SM0.0
LPS
A      传感器6:I0.5
AW<    T46, VW64
AW<    T106, +40
A      M1.3
A      I1.5
TON    T46, +600
LRD
AW>=   T46, +2
EU
+I     +1, VW62
LRD
A      T34
MOVW   +0, VW62
LPP
A      传感器6:I0.5
A      I1.5
A      M1.3
TON    T106, +40
END_SUBROUTINE_BLOCK

SUBROUTINE_BLOCK N7:SBR7
TITLE=
VAR_INPUT
连包长7:WORD;	// LW0 
屏地址7:BYTE;	// LB2 
报警袋数7:WORD;	// LW3 
END_VAR
VAR_OUTPUT
装车机7:BOOL;	// L5.0 
END_VAR
VAR
总袋数7:WORD;	// LW6 
袋长7:WORD;	// LW8 
已装袋数7:WORD;	// LW10 
剩余袋数7:WORD;	// LW12 
END_VAR
BEGIN
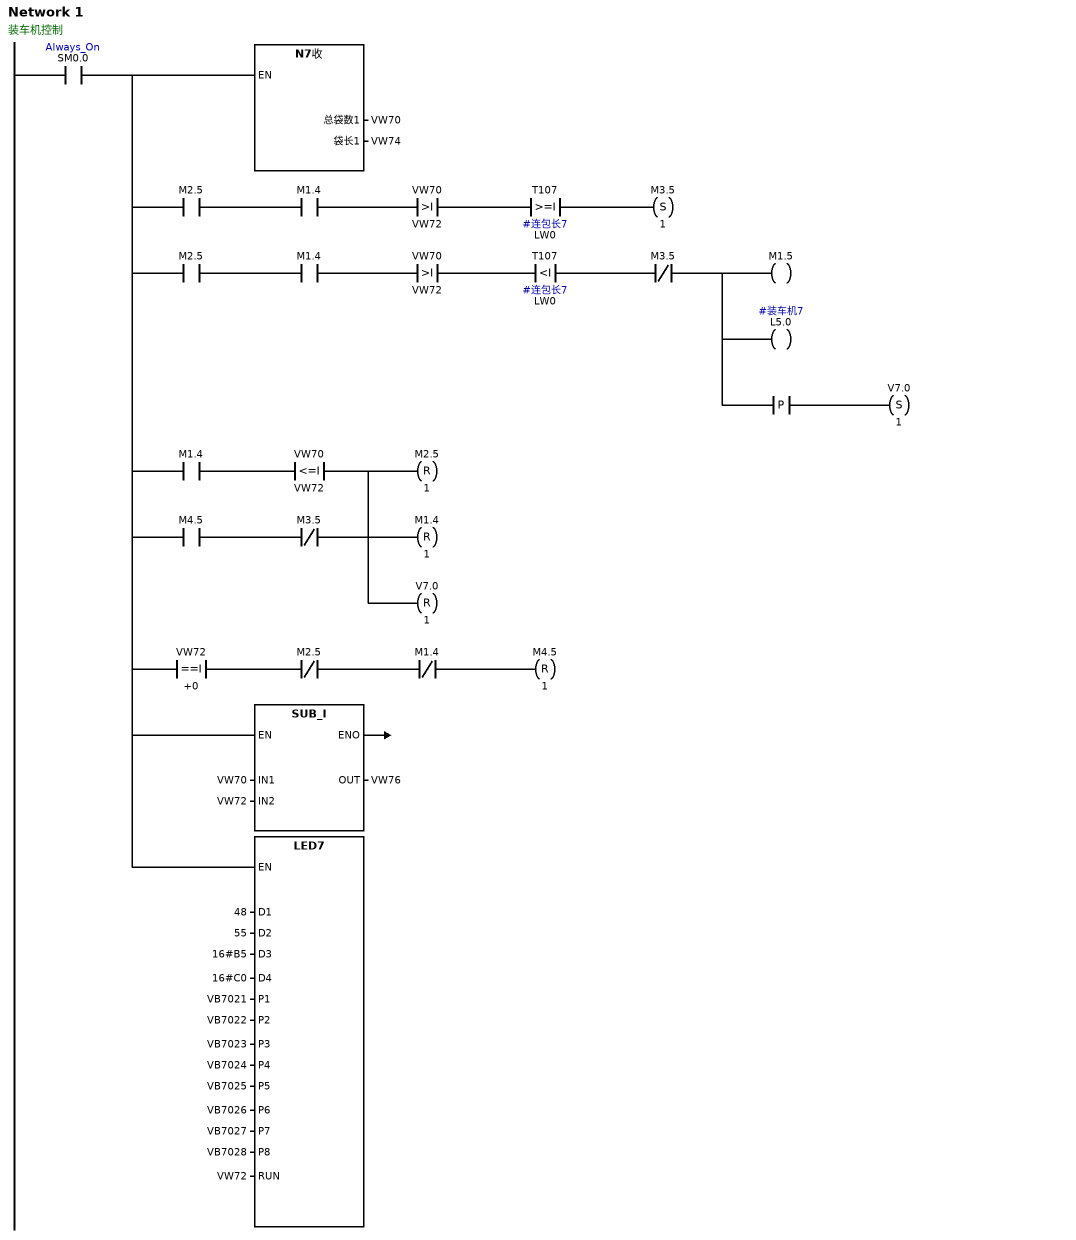
Network 1
// 装车机控制
LD     Always_On:SM0.0
LPS
CALL   N7收:SBR27, VW70, VW74
A      M2.5
A      M1.4
AW>    VW70, VW72
AW>=   T107, #连包长7:LW0
S      M3.5, 1
LRD
A      M2.5
A      M1.4
AW>    VW70, VW72
AW<    T107, #连包长7:LW0
AN     M3.5
=      M1.5
=      #装车机7:L5.0
EU
S      V7.0, 1
LRD
LD     M1.4
AW<=   VW70, VW72
LD     M4.5
AN     M3.5
OLD
ALD
R      M2.5, 1
R      M1.4, 1
R      V7.0, 1
LPP
LPS
AW=    VW72, +0
AN     M2.5
AN     M1.4
R      M4.5, 1
LRD
MOVW   VW70, VW76
-I     VW72, VW76
LPP
CALL   LED7:SBR17, 48, 55, 16#B5, 16#C0, VB7021, VB7022, VB7023, VB7024, VB7025, VB7026, VB7027, VB7028, VW72
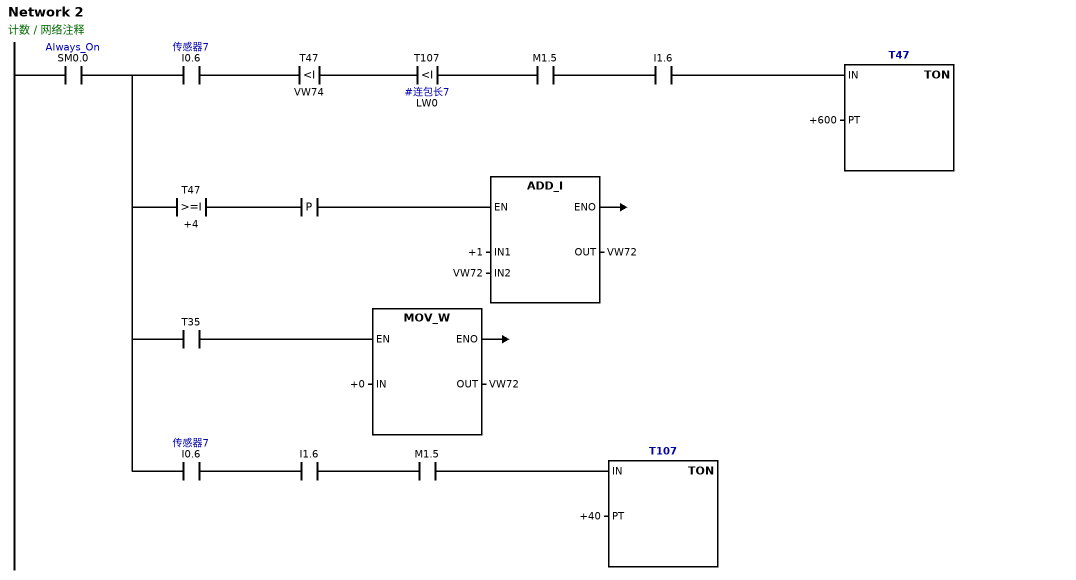
Network 2
// 计数
// 网络注释
LD     Always_On:SM0.0
LPS
A      传感器7:I0.6
AW<    T47, VW74
AW<    T107, #连包长7:LW0
A      M1.5
A      I1.6
TON    T47, +600
LRD
AW>=   T47, +4
EU
+I     +1, VW72
LRD
A      T35
MOVW   +0, VW72
LPP
A      传感器7:I0.6
A      I1.6
A      M1.5
TON    T107, +40
END_SUBROUTINE_BLOCK

SUBROUTINE_BLOCK N8:SBR8
TITLE=
VAR_INPUT
连包长8:WORD;	// LW0 
屏地址8:BYTE;	// LB2 
报警袋数8:WORD;	// LW3 
END_VAR
VAR_OUTPUT
装车机8:BOOL;	// L5.0 
END_VAR
VAR
总袋数8:WORD;	// LW6 
袋长8:WORD;	// LW8 
已装袋数8:WORD;	// LW10 
剩余袋数8:WORD;	// LW12 
END_VAR
BEGIN
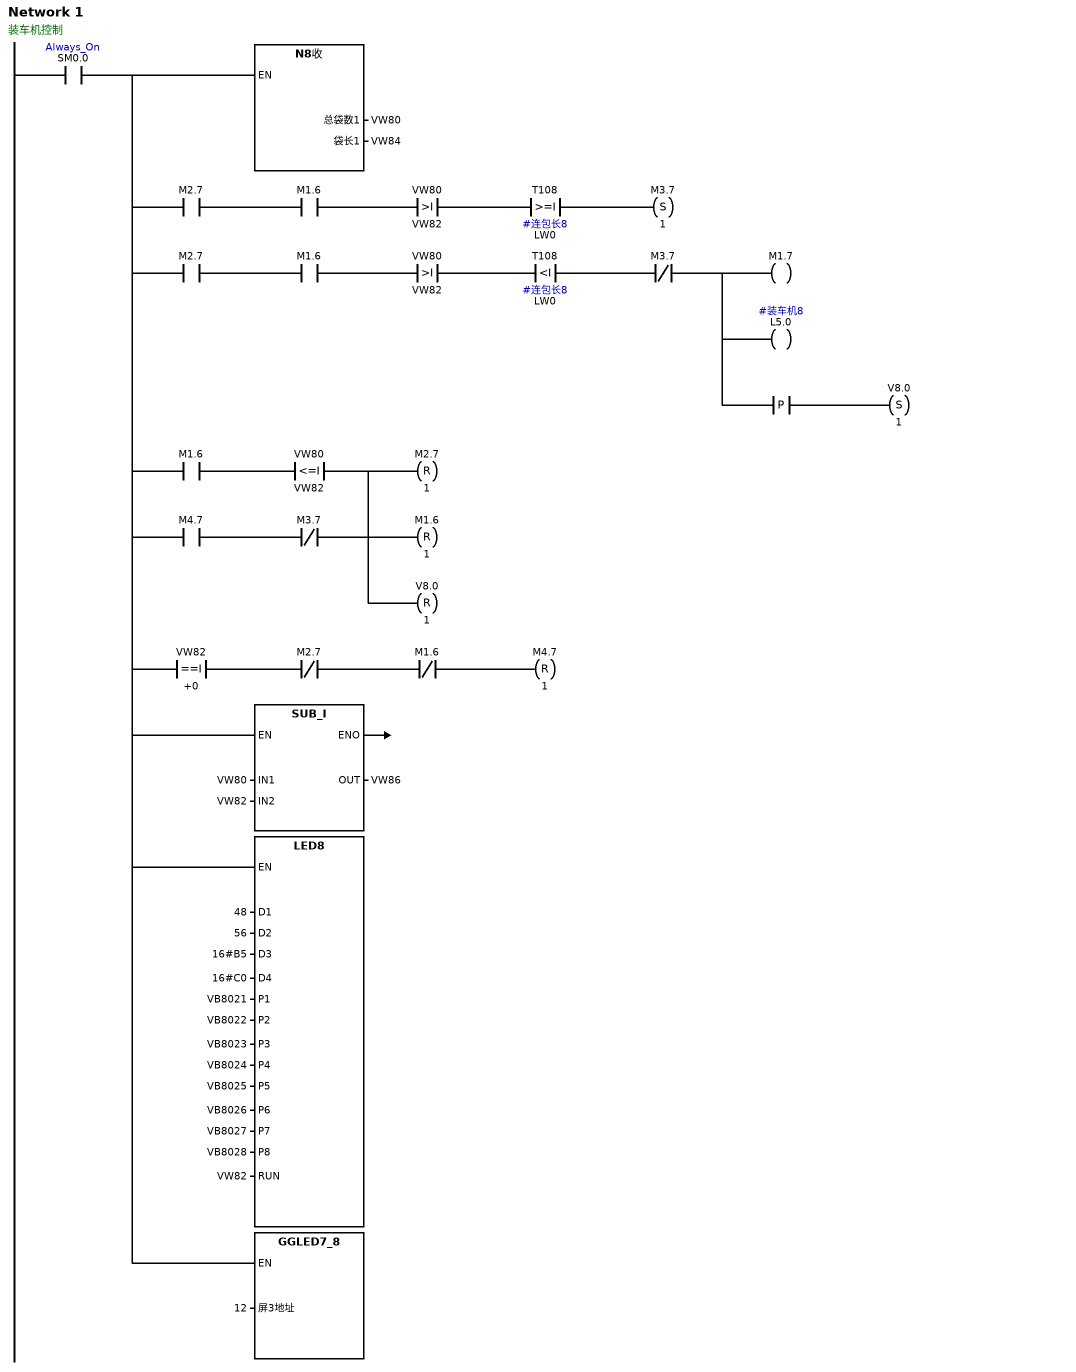
Network 1
// 装车机控制
LD     Always_On:SM0.0
LPS
CALL   N8收:SBR28, VW80, VW84
A      M2.7
A      M1.6
AW>    VW80, VW82
AW>=   T108, #连包长8:LW0
S      M3.7, 1
LRD
A      M2.7
A      M1.6
AW>    VW80, VW82
AW<    T108, #连包长8:LW0
AN     M3.7
=      M1.7
=      #装车机8:L5.0
EU
S      V8.0, 1
LRD
LD     M1.6
AW<=   VW80, VW82
LD     M4.7
AN     M3.7
OLD
ALD
R      M2.7, 1
R      M1.6, 1
R      V8.0, 1
LPP
LPS
AW=    VW82, +0
AN     M2.7
AN     M1.6
R      M4.7, 1
LRD
MOVW   VW80, VW86
-I     VW82, VW86
LRD
CALL   LED8:SBR18, 48, 56, 16#B5, 16#C0, VB8021, VB8022, VB8023, VB8024, VB8025, VB8026, VB8027, VB8028, VW82
LPP
CALL   GGLED7_8:SBR34, 12
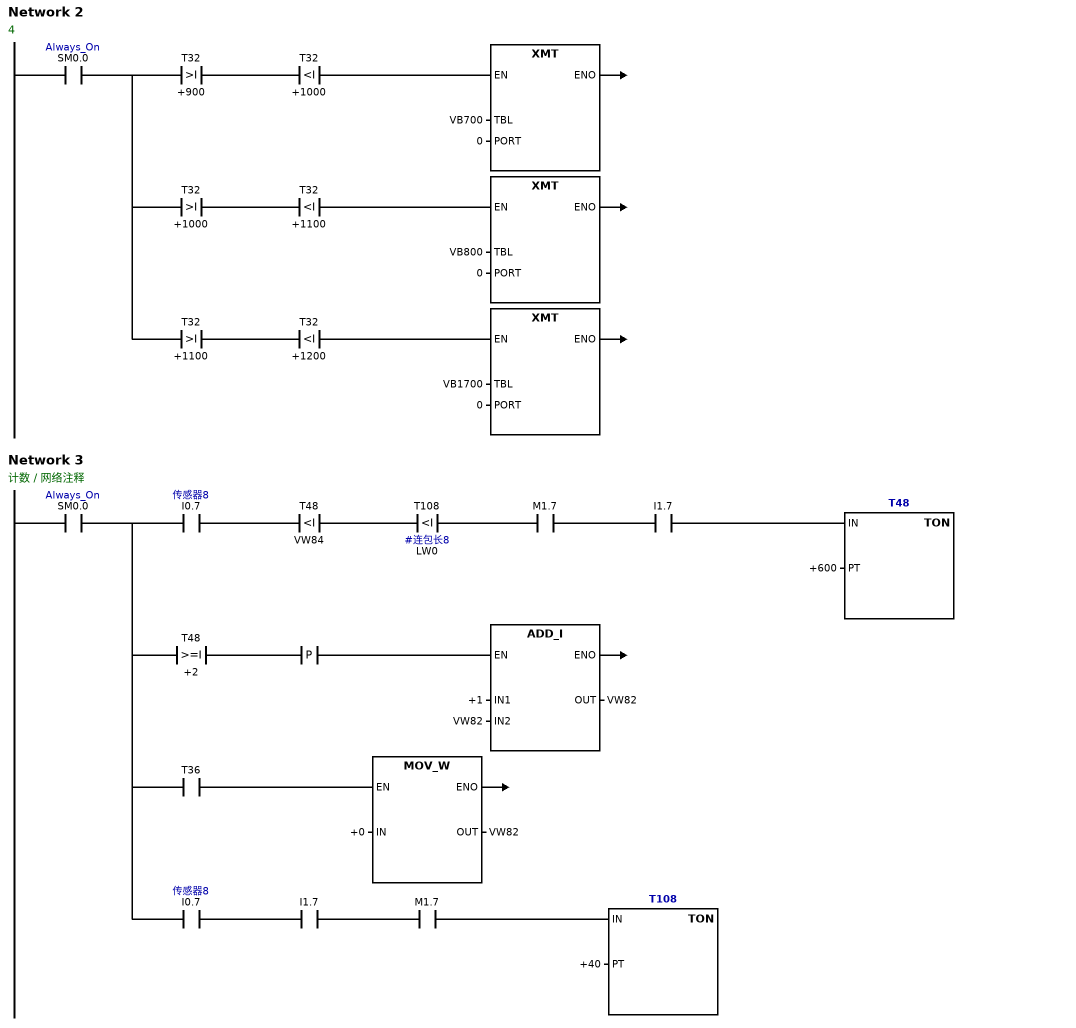
Network 2
// 4
LD     Always_On:SM0.0
LPS
AW>    T32, +900
AW<    T32, +1000
XMT    VB700, 0
LRD
AW>    T32, +1000
AW<    T32, +1100
XMT    VB800, 0
LPP
AW>    T32, +1100
AW<    T32, +1200
XMT    VB1700, 0
Network 3
// 计数
// 网络注释
LD     Always_On:SM0.0
LPS
A      传感器8:I0.7
AW<    T48, VW84
AW<    T108, #连包长8:LW0
A      M1.7
A      I1.7
TON    T48, +600
LRD
AW>=   T48, +2
EU
+I     +1, VW82
LRD
A      T36
MOVW   +0, VW82
LPP
A      传感器8:I0.7
A      I1.7
A      M1.7
TON    T108, +40
END_SUBROUTINE_BLOCK

// SBR9: protected block, not included

// SBR10: protected block, not included

SUBROUTINE_BLOCK LED1:SBR11
TITLE=
VAR_INPUT
D1:BYTE;	// LB0 
D2:BYTE;	// LB1 
D3:BYTE;	// LB2 
D4:BYTE;	// LB3 
P1:BYTE;	// LB4 
P2:BYTE;	// LB5 
P3:BYTE;	// LB6 
P4:BYTE;	// LB7 
P5:BYTE;	// LB8 
P6:BYTE;	// LB9 
P7:BYTE;	// LB10 
P8:BYTE;	// LB11 
RUN:WORD;	// LW12 
END_VAR
BEGIN
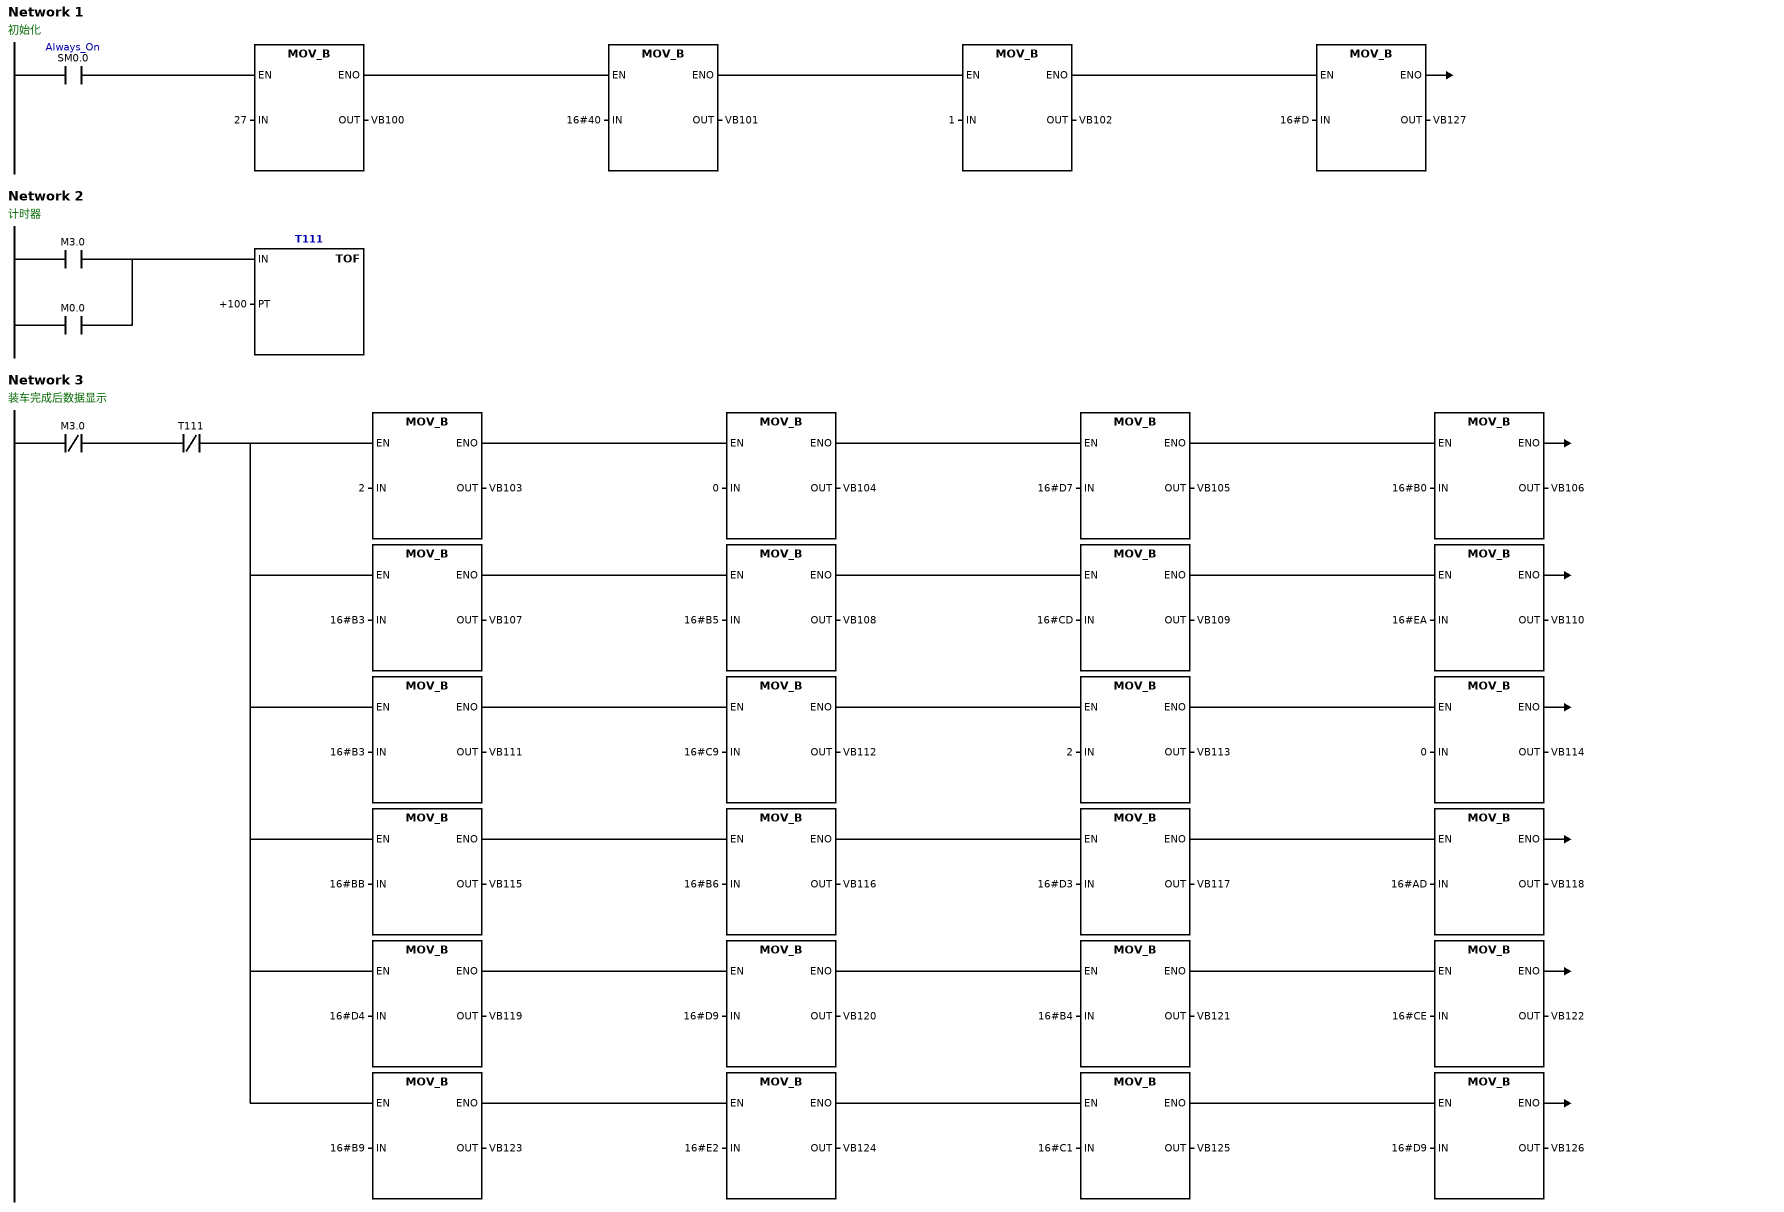
Network 1
// 初始化
LD     Always_On:SM0.0
MOVB   27, VB100
AENO
MOVB   16#40, VB101
AENO
MOVB   1, VB102
AENO
MOVB   16#D, VB127
Network 2
// 计时器
LD     M3.0
O      M0.0
TOF    T111, +100
Network 3
// 装车完成后数据显示
LDN    M3.0
AN     T111
LPS
MOVB   2, VB103
AENO
MOVB   0, VB104
AENO
MOVB   16#D7, VB105
AENO
MOVB   16#B0, VB106
LRD
MOVB   16#B3, VB107
AENO
MOVB   16#B5, VB108
AENO
MOVB   16#CD, VB109
AENO
MOVB   16#EA, VB110
LRD
MOVB   16#B3, VB111
AENO
MOVB   16#C9, VB112
AENO
MOVB   2, VB113
AENO
MOVB   0, VB114
LRD
MOVB   16#BB, VB115
AENO
MOVB   16#B6, VB116
AENO
MOVB   16#D3, VB117
AENO
MOVB   16#AD, VB118
LRD
MOVB   16#D4, VB119
AENO
MOVB   16#D9, VB120
AENO
MOVB   16#B4, VB121
AENO
MOVB   16#CE, VB122
LPP
MOVB   16#B9, VB123
AENO
MOVB   16#E2, VB124
AENO
MOVB   16#C1, VB125
AENO
MOVB   16#D9, VB126
